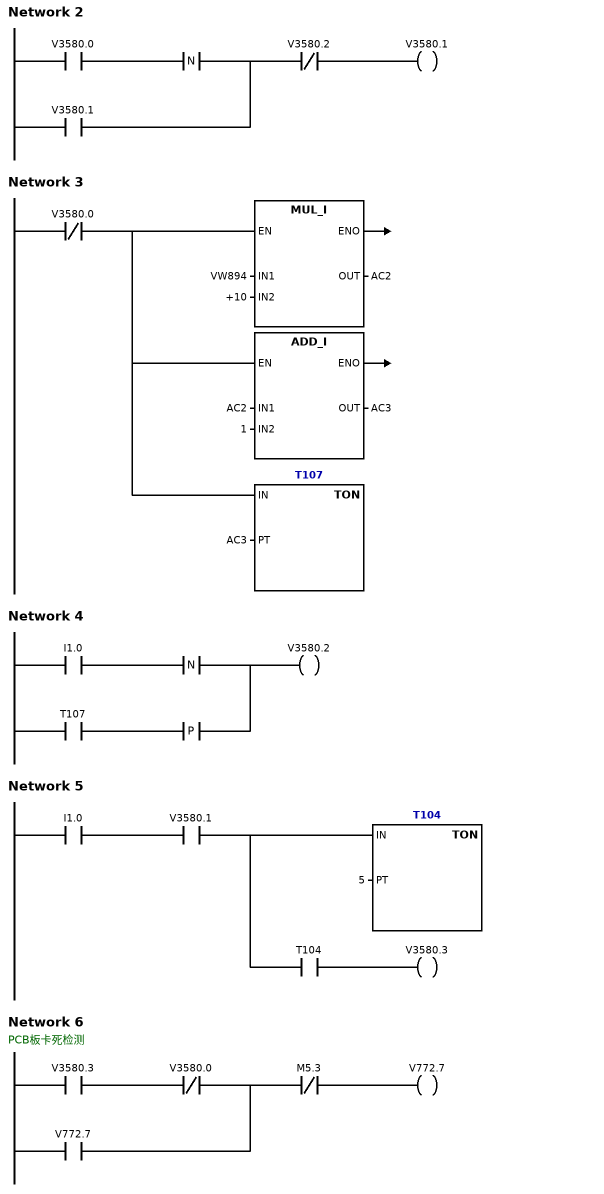
[picture p120: SBR45 networks 2-6]
Network 2
LD     V3580.0
ED
O      V3580.1
AN     V3580.2
=      V3580.1
Network 3
LDN    V3580.0
MOVW   VW894, AC2
*I     +10, AC2
MOVW   AC2, AC3
+I     1, AC3
TON    T107, AC3
Network 4
LD     I1.0
ED
LD     T107
EU
OLD
=      V3580.2
Network 5
LD     I1.0
A      V3580.1
TON    T104, 5
A      T104
=      V3580.3
Network 6
// PCB板卡死检测
LD     V3580.3
AN     V3580.0
O      V772.7
AN     M5.3
=      V772.7
Network 7 // 网络标题
// 网络注释
Network 17 // 网络标题
// 网络注释
Network 27 // Network Title
// Network Comment
Network 37 // 网络标题
// 网络注释
END_SUBROUTINE_BLOCK

SUBROUTINE_BLOCK programme_locked:SBR46
TITLE=子程序注释
BEGIN
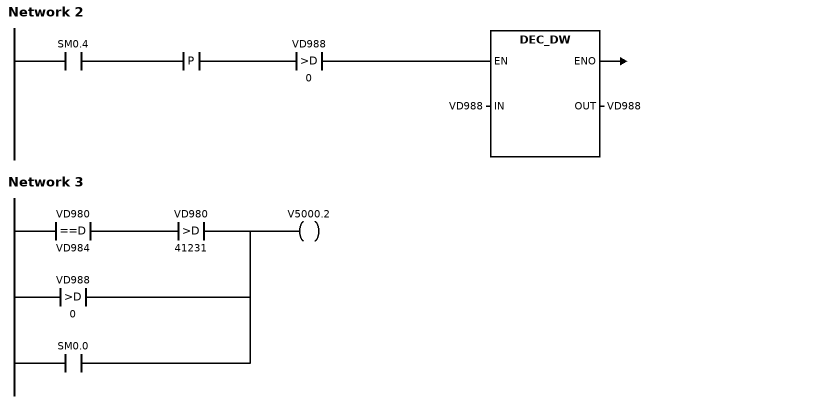
Network 2
LD     SM0.4
EU
AD>    VD988, 0
DECD   VD988
Network 3
LDD=   VD980, VD984
AD>    VD980, 41231
OD>    VD988, 0
O      SM0.0
=      V5000.2
Network 7 // 网络标题
// 网络注释
END_SUBROUTINE_BLOCK

// (further data pages could not be read)
